// Return CRC of the values stored in the dictionary.
FUNCTION F_DictionaryValuesCrc : WORD
VAR_IN_OUT
   Dictionary : FB_Dictionary;
END_VAR
VAR
   i : UDINT;
   sKey : T_MaxString;
   tValue : T_Arg;
END_VAR

IF Dictionary.Count > 0 THEN

   IF NOT Dictionary.TryGetIndex(Index := 0, Key := sKey, Value := tValue) THEN
      RETURN;
   ELSE
      F_DictionaryValuesCrc := F_DATA_TO_CRC16_CCITT(
         pData := tValue.pData,
         cbData := tValue.cbLen,
         crc := 16#FFFF // First pass needs the seed.
      );
   END_IF

END_IF

FOR i := 1 TO (Dictionary.Count - 1) DO

   IF NOT Dictionary.TryGetIndex(Index := 0, Key := sKey, Value := tValue) THEN
      F_DictionaryValuesCrc := 16#0000;
      RETURN;
   ELSE
      F_DictionaryValuesCrc := F_DATA_TO_CRC16_CCITT(
         pData := tValue.pData,
         cbData := tValue.cbLen,
         crc := F_DictionaryValuesCrc // iteratively pass in CRC.
      );
   END_IF

END_FOR

END_FUNCTION

(* stored: Version 1.1.0.1, ProductVersion 3.1.4024.9
   POU F_DictionaryValuesCrc: Id {35315de4-bb50-47a6-92c7-6ae3f8a96abc}, SpecialFunc None *)
